{attribute 'enable_dynamic_creation'}
FUNCTION_BLOCK FB_Circle IMPLEMENTS I_Shape
VAR_INPUT
END_VAR
VAR_OUTPUT
END_VAR
VAR
END_VAR

//Agregue el {atributo 'enable_dynamic_creation'} en la parte superior de la sección de declaración de cada bloque de funciones. 
//Esto nos permitirá crear una instancia de cada bloque de funciones dinámicamente usando el operador _NEW en el bloque de funciones FB_ShapeCreator.

METHOD M_Draw : BOOL
ADSLOGSTR(ADSLOG_MSGTYPE_HINT, 'Draw circle', '');
M_Draw := TRUE;
END_METHOD

END_FUNCTION_BLOCK

(* stored: Version 1.1.0.1, ProductVersion 3.1.4024.12
   POU FB_Circle: Id {b0f1baba-fd54-439d-972f-c8b3bbe19832}, SpecialFunc None
   Method M_Draw: Id {f6c025cf-fb05-4801-af03-76afb31347dd} *)
